# EPICS substitutions: TPGSup/TPG300_function_statuses.substitutions
file TPG300_function_statuses.template {

pattern {PORT, P, Q}
{"\$(PORT)", "\$(P)", "1"}
{"\$(PORT)", "\$(P)", "2"}
{"\$(PORT)", "\$(P)", "3"}
{"\$(PORT)", "\$(P)", "4"}

}
